TEXTLIST WorkAreaYesNo
  0 = 'No'
  1 = 'Yes'
   = ''
END_TEXTLIST

(* stored: Version 1.1.0.1, ProductVersion 3.1.4024.11
   TextList WorkAreaYesNo: Id {a1584761-c0a5-405d-802d-1d971af901f4} *)
